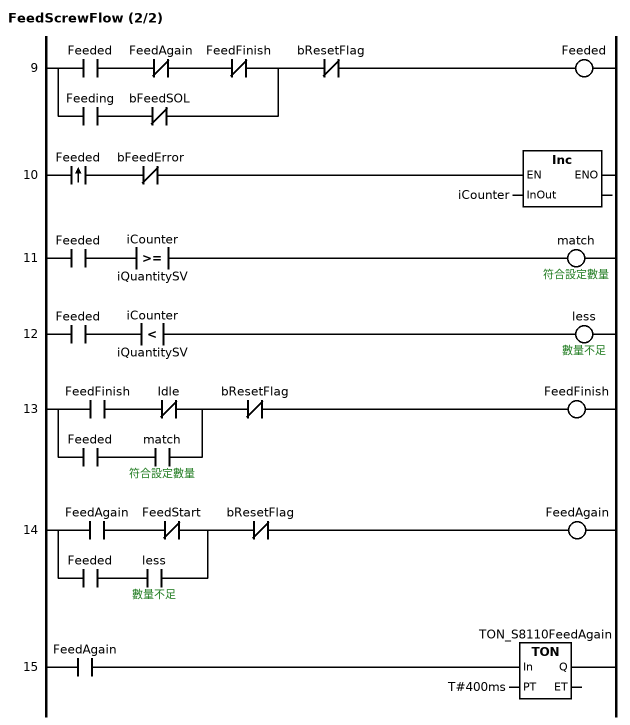
(* [picture p24: FeedScrewFlow, rungs 9-15] *)
(* Rung 9 *)
Feeded := ((Feeded AND NOT FeedAgain AND NOT FeedFinish) OR (Feeding AND NOT bFeedSOL)) AND NOT bResetFlag;
(* Rung 10 *)
_e2(CLK := Feeded);
IF _e2.Q AND NOT bFeedError THEN Inc(InOut := iCounter); END_IF;
(* Rung 11 *)
match := Feeded AND (iCounter >= iQuantitySV);
(* Rung 12 *)
less := Feeded AND (iCounter < iQuantitySV);
(* Rung 13 *)
FeedFinish := ((FeedFinish AND NOT Idle) OR (Feeded AND match)) AND NOT bResetFlag;
(* Rung 14 *)
FeedAgain := ((FeedAgain AND NOT FeedStart) OR (Feeded AND less)) AND NOT bResetFlag;
(* Rung 15 *)
TON_S8110FeedAgain(In := FeedAgain, PT := T#400ms);
END_FUNCTION_BLOCK

FUNCTION_BLOCK StanleyScrewFlow
VAR
    TON_PON : TON;
    PowerOn : BOOL;
    TON_PowerOn : TON;
    Idle : BOOL;
    ScrewStart : BOOL;
    Screwing : BOOL;
    Screwed : BOOL;
    ScrewAgain : BOOL;
    ScrewFinish : BOOL;
    ClearCount : BOOL;
    match : BOOL;  (* 符合設定數量 *)
    less : BOOL;  (* 數量不足 *)
    TON_S8110FeedAgain : TON;
    screwokstatus : BOOL;
    screwnokstatus : BOOL;
END_VAR
VAR_OUTPUT
    bOKFlag : BOOL;
    bNGFlag : BOOL;
END_VAR
VAR_INPUT
    ENABLE : BOOL;
    bStratFlag : BOOL;
    bResetFlag : BOOL;
    bErrorStatus : BOOL;
    bScrewNOK : BOOL;
    bScrewOK : BOOL;
    bScrewInCycle : BOOL;
    iQuantitySV : INT;
END_VAR
VAR_IN_OUT
    iCounter : INT;
END_VAR
VAR
    _e1 : R_TRIG;
    _e2 : R_TRIG;
    _e3 : R_TRIG;
    _e4 : R_TRIG;
END_VAR
(* ladder, written here as Structured Text *)

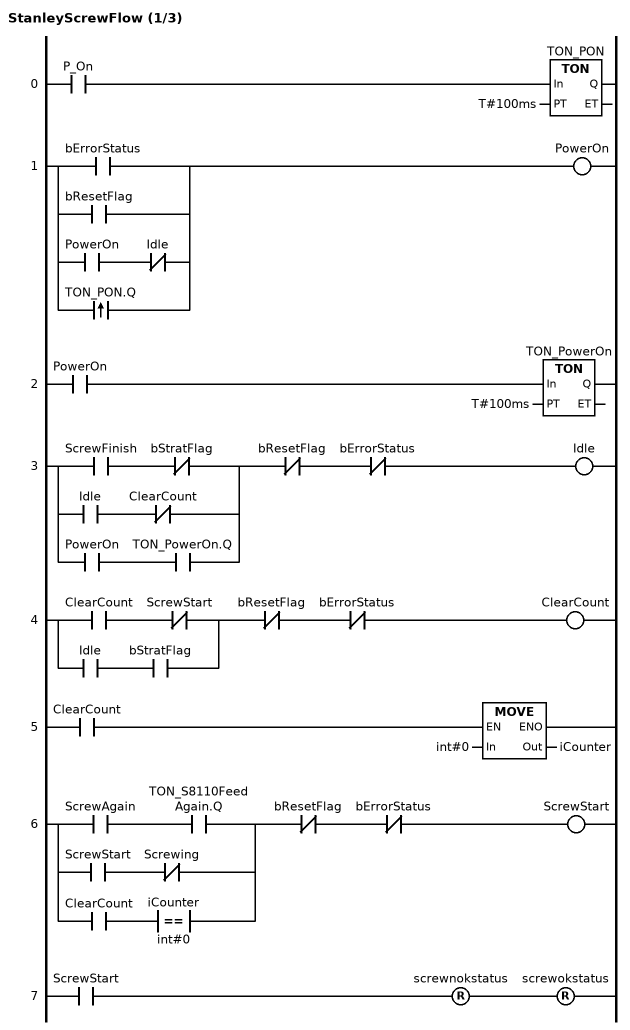
(* Rung 0 *)
TON_PON(In := P_On, PT := T#100ms);
(* Rung 1 *)
_e1(CLK := TON_PON.Q);
PowerOn := bErrorStatus OR bResetFlag OR (PowerOn AND NOT Idle) OR _e1.Q;
(* Rung 2 *)
TON_PowerOn(In := PowerOn, PT := T#100ms);
(* Rung 3 *)
Idle := ((ScrewFinish AND NOT bStratFlag) OR (Idle AND NOT ClearCount) OR (PowerOn AND TON_PowerOn.Q)) AND NOT bResetFlag AND NOT bErrorStatus;
(* Rung 4 *)
ClearCount := ((ClearCount AND NOT ScrewStart) OR (Idle AND bStratFlag)) AND NOT bResetFlag AND NOT bErrorStatus;
(* Rung 5 *)
IF ClearCount THEN iCounter := int#0; END_IF;
(* Rung 6 *)
ScrewStart := ((ScrewAgain AND TON_S8110FeedAgain.Q) OR (ScrewStart AND NOT Screwing) OR (ClearCount AND (iCounter = int#0))) AND NOT bResetFlag AND NOT bErrorStatus;
(* Rung 7 *)
IF ScrewStart THEN
    screwnokstatus := FALSE;
    screwokstatus := FALSE;
END_IF;

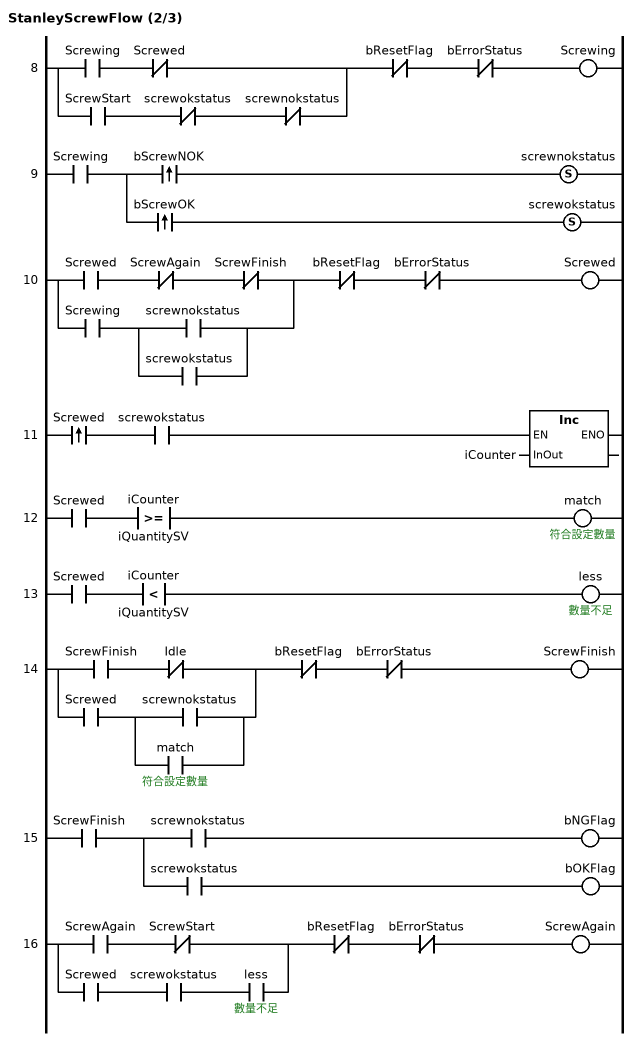
(* Rung 8 *)
Screwing := ((Screwing AND NOT Screwed) OR (ScrewStart AND NOT screwokstatus AND NOT screwnokstatus)) AND NOT bResetFlag AND NOT bErrorStatus;
(* Rung 9 *)
_e2(CLK := bScrewNOK);
IF Screwing AND _e2.Q THEN screwnokstatus := TRUE; END_IF;
_e3(CLK := bScrewOK);
IF Screwing AND _e3.Q THEN screwokstatus := TRUE; END_IF;
(* Rung 10 *)
Screwed := ((Screwed AND NOT ScrewAgain AND NOT ScrewFinish) OR (Screwing AND (screwnokstatus OR screwokstatus))) AND NOT bResetFlag AND NOT bErrorStatus;
(* Rung 11 *)
_e4(CLK := Screwed);
IF _e4.Q AND screwokstatus THEN Inc(InOut := iCounter); END_IF;
(* Rung 12 *)
match := Screwed AND (iCounter >= iQuantitySV);
(* Rung 13 *)
less := Screwed AND (iCounter < iQuantitySV);
(* Rung 14 *)
ScrewFinish := ((ScrewFinish AND NOT Idle) OR (Screwed AND (screwnokstatus OR match))) AND NOT bResetFlag AND NOT bErrorStatus;
(* Rung 15 *)
bNGFlag := ScrewFinish AND screwnokstatus;
bOKFlag := ScrewFinish AND screwokstatus;
(* Rung 16 *)
ScrewAgain := ((ScrewAgain AND NOT ScrewStart) OR (Screwed AND screwokstatus AND less)) AND NOT bResetFlag AND NOT bErrorStatus;

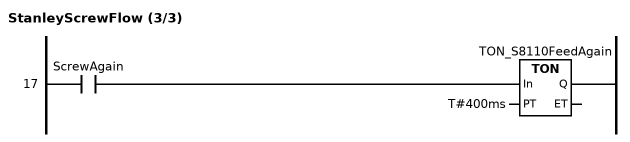
(* Rung 17 *)
TON_S8110FeedAgain(In := ScrewAgain, PT := T#400ms);
END_FUNCTION_BLOCK

FUNCTION_BLOCK StanleyJobSelect
VAR_INPUT
    Enable : BOOL;
    iJobNo : INT;
END_VAR
VAR_OUTPUT
    bJobBit0 : BOOL;
    bJobBit1 : BOOL;
    bJobBit2 : BOOL;
END_VAR
CASE iJobNo OF
    0 : 	bJobBit0:=FALSE;
			bJobBit1 :=FALSE;
			bJobBit2:=FALSE;
			
    1 : 	bJobBit0:=TRUE;
			bJobBit1:=FALSE;
			bJobBit2:=FALSE;
			
    2 : 	bJobBit0:=FALSE;
			bJobBit1:=TRUE;
			bJobBit2:=FALSE;
			
    3 : 	bJobBit0:=TRUE;
			bJobBit1:=TRUE;
			bJobBit2:=FALSE;
			
    4 : 	bJobBit0:=FALSE;
			bJobBit1:=FALSE;
			bJobBit2:=TRUE;
			
    5 : 	bJobBit0:=TRUE;
			bJobBit1:=FALSE;
			bJobBit2:=TRUE;
			
    6 : 	bJobBit0:=FALSE;
			bJobBit1:=TRUE;
			bJobBit2:=TRUE;
			
    7 : 	bJobBit0:=TRUE;
			bJobBit1:=TRUE;
			bJobBit2:=TRUE;
ELSE
    bJobBit0:=FALSE;
	bJobBit1:=FALSE;
	bJobBit2:=FALSE;
END_CASE;
END_FUNCTION_BLOCK

FUNCTION_BLOCK CCD
VAR
    TON_PON : TON;
    TON_PowerOn : TON;
    TON_CCDStart : TON;
    TON_CCDStarting : TON;
    TON_CCDFinish : TON;
    PowerOn : BOOL;
    Idle : BOOL;
    CCDStart : BOOL;
    CCDStarting : BOOL;
    CCDFinish : BOOL;
    SetFlagFinish : BOOL;
    iCounter : INT;
    ECErrorReset : ResetECError;
END_VAR
VAR_INPUT
    Enable : BOOL;
    bCCDReady : BOOL;
    bResetFlag : BOOL;
    bStratFlag : BOOL;
    bCCDStartPB : BOOL;
    diCCDokFlag : DINT;
    diCCDngFlag : DINT;
END_VAR
VAR_OUTPUT
    bCCDTrigger : BOOL;
    bErrorFlag : BOOL;
END_VAR
VAR_IN_OUT
    bOKFlag : BOOL;
    bNGFlag : BOOL;
END_VAR
VAR_INPUT
    bCCDBusy : BOOL;
END_VAR
VAR
    _e1 : R_TRIG;
    _e2 : R_TRIG;
END_VAR
(* ladder, written here as Structured Text *)

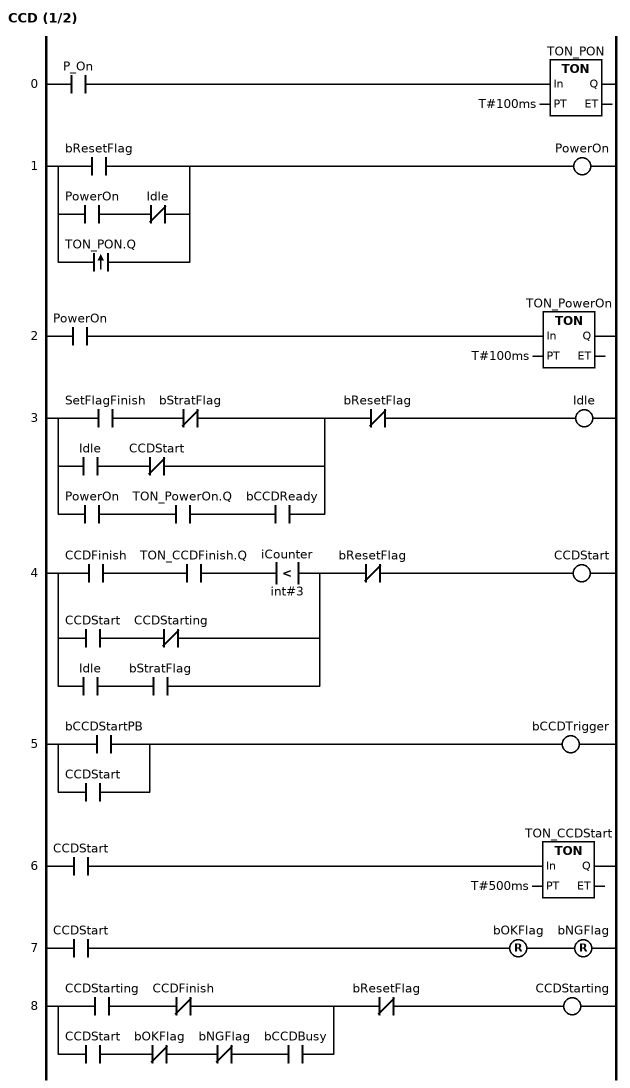
(* Rung 0 *)
TON_PON(In := P_On, PT := T#100ms);
(* Rung 1 *)
_e1(CLK := TON_PON.Q);
PowerOn := bResetFlag OR (PowerOn AND NOT Idle) OR _e1.Q;
(* Rung 2 *)
TON_PowerOn(In := PowerOn, PT := T#100ms);
(* Rung 3 *)
Idle := ((SetFlagFinish AND NOT bStratFlag) OR (Idle AND NOT CCDStart) OR (PowerOn AND TON_PowerOn.Q AND bCCDReady)) AND NOT bResetFlag;
(* Rung 4 *)
CCDStart := ((CCDFinish AND TON_CCDFinish.Q AND (iCounter < int#3)) OR (CCDStart AND NOT CCDStarting) OR (Idle AND bStratFlag)) AND NOT bResetFlag;
(* Rung 5 *)
bCCDTrigger := bCCDStartPB OR CCDStart;
(* Rung 6 *)
TON_CCDStart(In := CCDStart, PT := T#500ms);
(* Rung 7 *)
IF CCDStart THEN
    bOKFlag := FALSE;
    bNGFlag := FALSE;
END_IF;
(* Rung 8 *)
CCDStarting := ((CCDStarting AND NOT CCDFinish) OR (CCDStart AND NOT bOKFlag AND NOT bNGFlag AND bCCDBusy)) AND NOT bResetFlag;

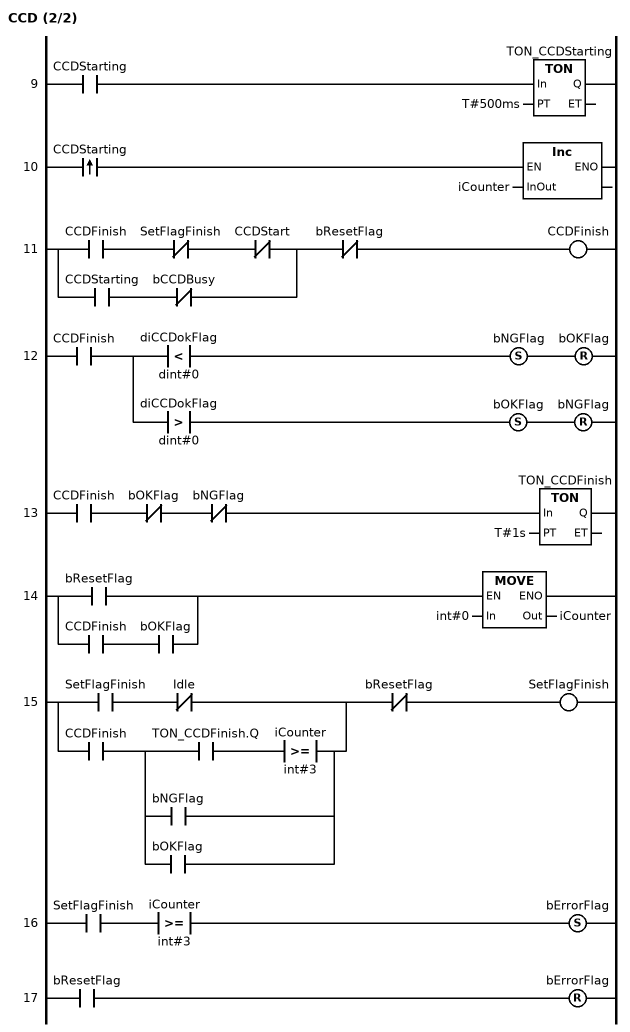
(* Rung 9 *)
TON_CCDStarting(In := CCDStarting, PT := T#500ms);
(* Rung 10 *)
_e2(CLK := CCDStarting);
IF _e2.Q THEN Inc(InOut := iCounter); END_IF;
(* Rung 11 *)
CCDFinish := ((CCDFinish AND NOT SetFlagFinish AND NOT CCDStart) OR (CCDStarting AND NOT bCCDBusy)) AND NOT bResetFlag;
(* Rung 12 *)
IF CCDFinish AND (diCCDokFlag < dint#0) THEN
    bNGFlag := TRUE;
    bOKFlag := FALSE;
END_IF;
IF CCDFinish AND (diCCDokFlag > dint#0) THEN
    bOKFlag := TRUE;
    bNGFlag := FALSE;
END_IF;
(* Rung 13 *)
TON_CCDFinish(In := CCDFinish AND NOT bOKFlag AND NOT bNGFlag, PT := T#1s);
(* Rung 14 *)
IF bResetFlag OR (CCDFinish AND bOKFlag) THEN iCounter := int#0; END_IF;
(* Rung 15 *)
SetFlagFinish := ((SetFlagFinish AND NOT Idle) OR (CCDFinish AND ((TON_CCDFinish.Q AND (iCounter >= int#3)) OR bNGFlag OR bOKFlag))) AND NOT bResetFlag;
(* Rung 16 *)
IF SetFlagFinish AND (iCounter >= int#3) THEN bErrorFlag := TRUE; END_IF;
(* Rung 17 *)
IF bResetFlag THEN bErrorFlag := FALSE; END_IF;
END_FUNCTION_BLOCK

FUNCTION_BLOCK Station_1Step
VAR
    timer_PON : TON;
    PowerOn : BOOL;
    Idle : BOOL;
    Step1Start : BOOL;
    Step1Running : BOOL;
    Step1Finish : BOOL;
END_VAR
VAR_OUTPUT
    outStep1StartFlag : BOOL;
    inoutCurrentStationWork : BOOL;
END_VAR
VAR_INPUT
    Enable : BOOL;
    inAutoStatus : BOOL;
    inResetFlag : BOOL;
    inErrorStatus : BOOL;
    inEnablePB : BOOL;
    inMachineStart : BOOL;
    inExStationFinish : BOOL;
    inExStationOK : BOOL;
    inExStationNG : BOOL;
    inStep1FinishFlag : BOOL;
END_VAR
VAR_IN_OUT
    inoutCurrentStationFinish : BOOL;
    inoutCurrentStationOK : BOOL;
    inoutCurrentStationNG : BOOL;
END_VAR
VAR
    _e1 : R_TRIG;
END_VAR
(* ladder, written here as Structured Text *)

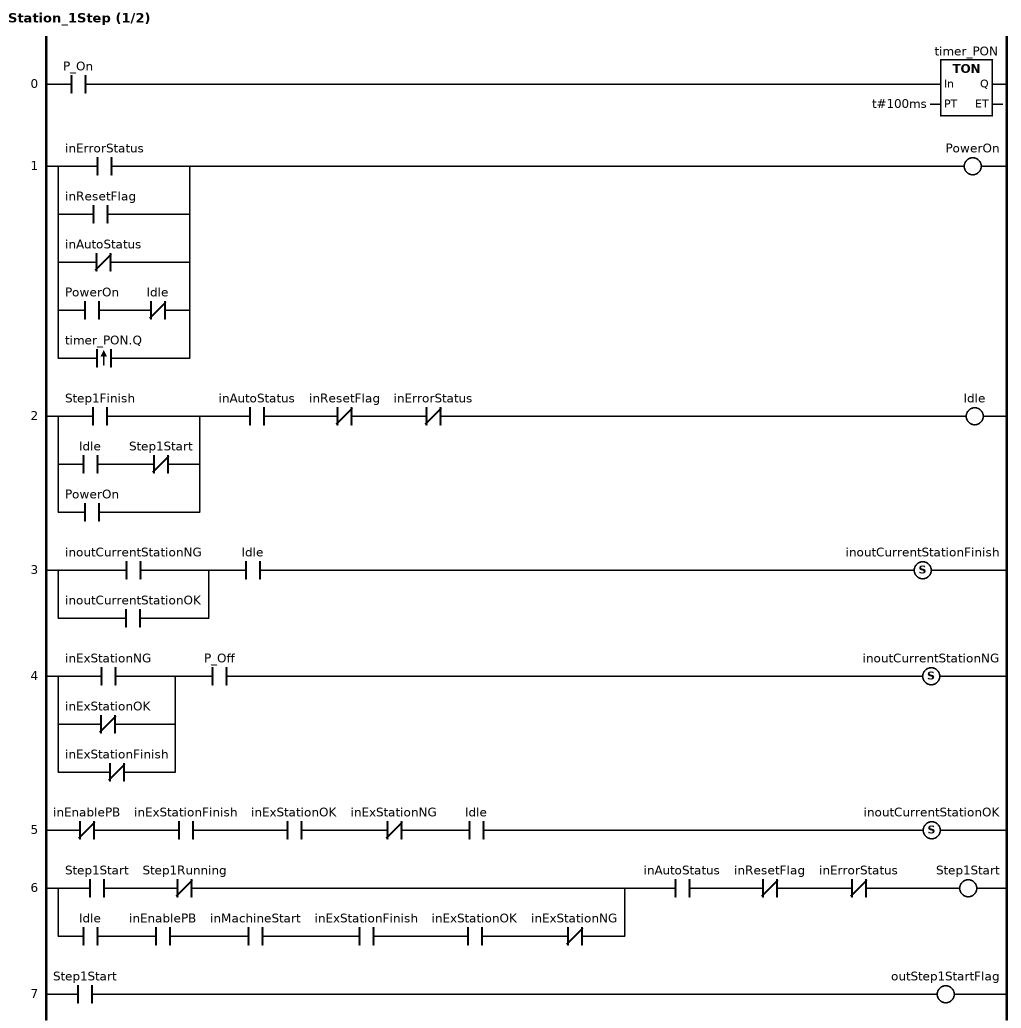
(* Rung 0 *)
timer_PON(In := P_On, PT := t#100ms);
(* Rung 1 *)
_e1(CLK := timer_PON.Q);
PowerOn := inErrorStatus OR inResetFlag OR NOT inAutoStatus OR (PowerOn AND NOT Idle) OR _e1.Q;
(* Rung 2 *)
Idle := (Step1Finish OR (Idle AND NOT Step1Start) OR PowerOn) AND inAutoStatus AND NOT inResetFlag AND NOT inErrorStatus;
(* Rung 3 *)
IF (inoutCurrentStationNG OR inoutCurrentStationOK) AND Idle THEN
    inoutCurrentStationFinish := TRUE;
END_IF;
(* Rung 4 *)
IF (inExStationNG OR NOT inExStationOK OR NOT inExStationFinish) AND P_Off THEN
    inoutCurrentStationNG := TRUE;
END_IF;
(* Rung 5 *)
IF NOT inEnablePB AND inExStationFinish AND inExStationOK AND NOT inExStationNG AND Idle THEN
    inoutCurrentStationOK := TRUE;
END_IF;
(* Rung 6 *)
Step1Start := ((Step1Start AND NOT Step1Running) OR (Idle AND inEnablePB AND inMachineStart AND inExStationFinish AND inExStationOK AND NOT inExStationNG)) AND inAutoStatus AND NOT inResetFlag AND NOT inErrorStatus;
(* Rung 7 *)
outStep1StartFlag := Step1Start;

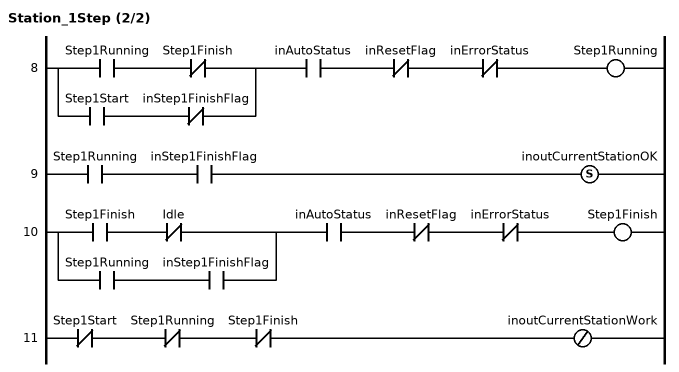
(* Rung 8 *)
Step1Running := ((Step1Running AND NOT Step1Finish) OR (Step1Start AND NOT inStep1FinishFlag)) AND inAutoStatus AND NOT inResetFlag AND NOT inErrorStatus;
(* Rung 9 *)
IF Step1Running AND inStep1FinishFlag THEN inoutCurrentStationOK := TRUE; END_IF;
(* Rung 10 *)
Step1Finish := ((Step1Finish AND NOT Idle) OR (Step1Running AND inStep1FinishFlag)) AND inAutoStatus AND NOT inResetFlag AND NOT inErrorStatus;
(* Rung 11 *)
inoutCurrentStationWork := NOT (NOT Step1Start AND NOT Step1Running AND NOT Step1Finish);
END_FUNCTION_BLOCK

FUNCTION_BLOCK Station_2Step
VAR
    timer_PON : TON;
    PowerOn : BOOL;
    Idle : BOOL;
    Step1Start : BOOL;
    Step1Running : BOOL;
    Step1Finish : BOOL;
    Step2Start : BOOL;
    Step2Running : BOOL;
    Step2Finish : BOOL;
END_VAR
VAR_OUTPUT
    outStep1StartFlag : BOOL;
    outStep2StartFlag : BOOL;
    inoutCurrentStationWork : BOOL;
END_VAR
VAR_INPUT
    Enable : BOOL;
    inAutoStatus : BOOL;
    inResetFlag : BOOL;
    inErrorStatus : BOOL;
    inEnablePB : BOOL;
    inMachineStart : BOOL;
    inExStationFinish : BOOL;
    inExStationOK : BOOL;
    inExStationNG : BOOL;
    inStep1FinishFlag : BOOL;
    inStep2OKFlag : BOOL;
    inStep2NGFlag : BOOL;
END_VAR
VAR_IN_OUT
    inoutCurrentStationFinish : BOOL;
    inoutCurrentStationOK : BOOL;
    inoutCurrentStationNG : BOOL;
END_VAR
VAR
    _e1 : R_TRIG;
END_VAR
(* ladder, written here as Structured Text *)

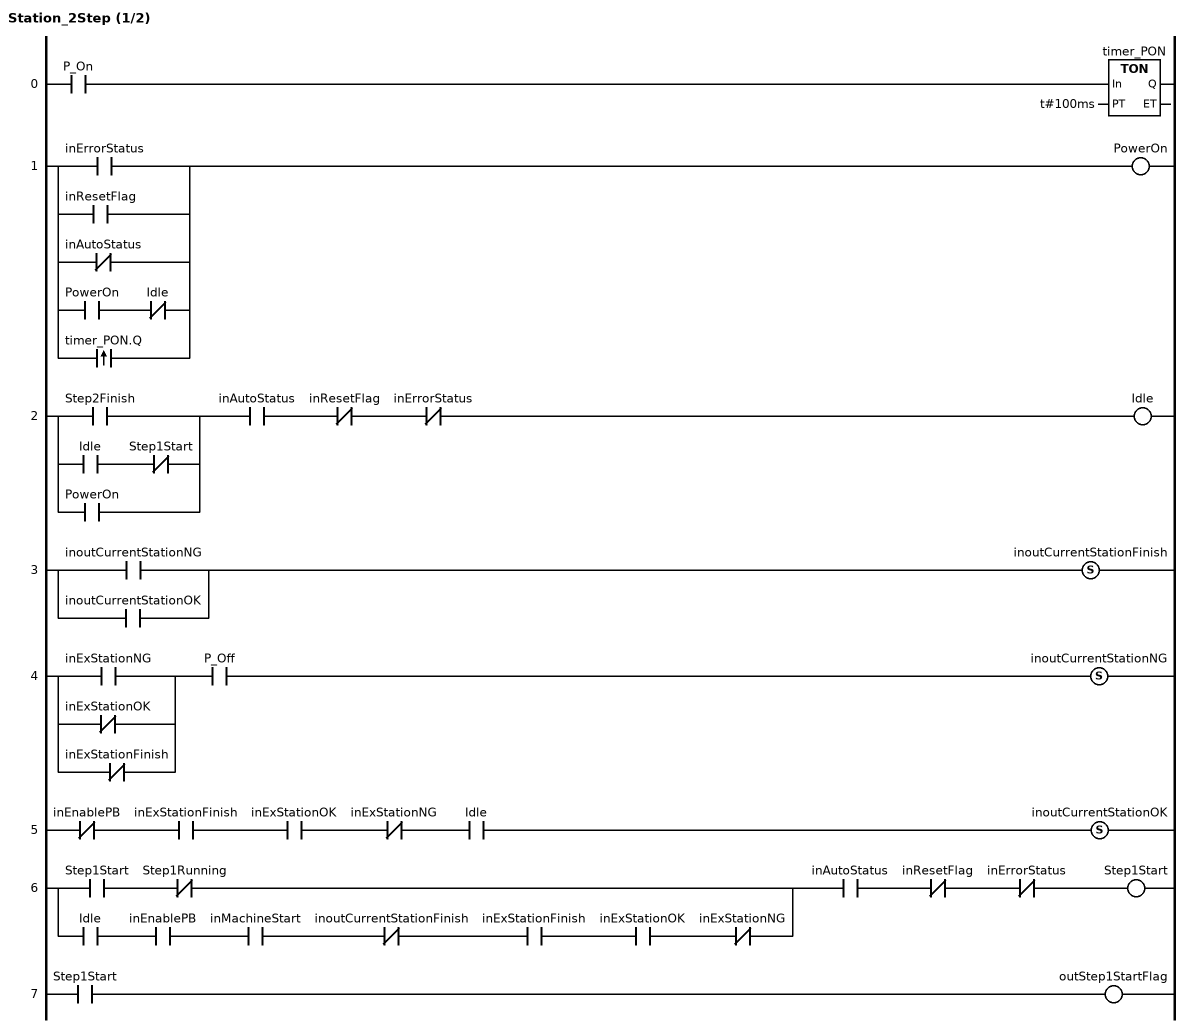
(* Rung 0 *)
timer_PON(In := P_On, PT := t#100ms);
(* Rung 1 *)
_e1(CLK := timer_PON.Q);
PowerOn := inErrorStatus OR inResetFlag OR NOT inAutoStatus OR (PowerOn AND NOT Idle) OR _e1.Q;
(* Rung 2 *)
Idle := (Step2Finish OR (Idle AND NOT Step1Start) OR PowerOn) AND inAutoStatus AND NOT inResetFlag AND NOT inErrorStatus;
(* Rung 3 *)
IF inoutCurrentStationNG OR inoutCurrentStationOK THEN inoutCurrentStationFinish := TRUE; END_IF;
(* Rung 4 *)
IF (inExStationNG OR NOT inExStationOK OR NOT inExStationFinish) AND P_Off THEN
    inoutCurrentStationNG := TRUE;
END_IF;
(* Rung 5 *)
IF NOT inEnablePB AND inExStationFinish AND inExStationOK AND NOT inExStationNG AND Idle THEN
    inoutCurrentStationOK := TRUE;
END_IF;
(* Rung 6 *)
Step1Start := ((Step1Start AND NOT Step1Running) OR (Idle AND inEnablePB AND inMachineStart AND NOT inoutCurrentStationFinish AND inExStationFinish AND inExStationOK AND NOT inExStationNG)) AND inAutoStatus AND NOT inResetFlag AND NOT inErrorStatus;
(* Rung 7 *)
outStep1StartFlag := Step1Start;

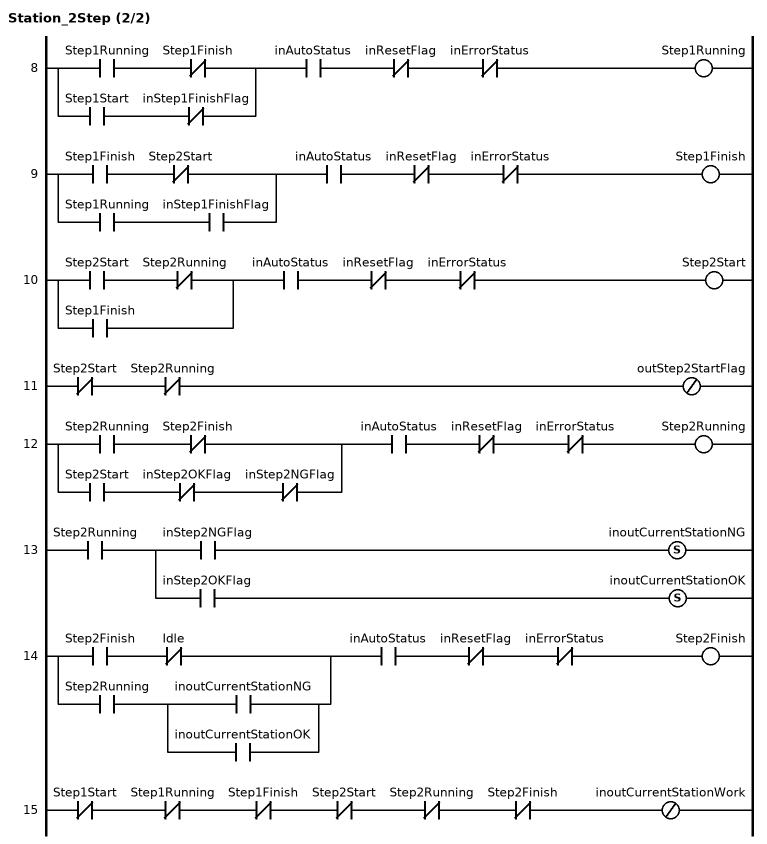
(* Rung 8 *)
Step1Running := ((Step1Running AND NOT Step1Finish) OR (Step1Start AND NOT inStep1FinishFlag)) AND inAutoStatus AND NOT inResetFlag AND NOT inErrorStatus;
(* Rung 9 *)
Step1Finish := ((Step1Finish AND NOT Step2Start) OR (Step1Running AND inStep1FinishFlag)) AND inAutoStatus AND NOT inResetFlag AND NOT inErrorStatus;
(* Rung 10 *)
Step2Start := ((Step2Start AND NOT Step2Running) OR Step1Finish) AND inAutoStatus AND NOT inResetFlag AND NOT inErrorStatus;
(* Rung 11 *)
outStep2StartFlag := NOT (NOT Step2Start AND NOT Step2Running);
(* Rung 12 *)
Step2Running := ((Step2Running AND NOT Step2Finish) OR (Step2Start AND NOT inStep2OKFlag AND NOT inStep2NGFlag)) AND inAutoStatus AND NOT inResetFlag AND NOT inErrorStatus;
(* Rung 13 *)
IF Step2Running AND inStep2NGFlag THEN inoutCurrentStationNG := TRUE; END_IF;
IF Step2Running AND inStep2OKFlag THEN inoutCurrentStationOK := TRUE; END_IF;
(* Rung 14 *)
Step2Finish := ((Step2Finish AND NOT Idle) OR (Step2Running AND (inoutCurrentStationNG OR inoutCurrentStationOK))) AND inAutoStatus AND NOT inResetFlag AND NOT inErrorStatus;
(* Rung 15 *)
inoutCurrentStationWork := NOT (NOT Step1Start AND NOT Step1Running AND NOT Step1Finish AND NOT Step2Start AND NOT Step2Running AND NOT Step2Finish);
END_FUNCTION_BLOCK